Omron CX-Programmer project NewProject (CX-Programmer 9.51)

# PLC NewPLC1: CP1H XA

## Global symbols (name address type ; comment)
10.00 BOOL  ; internal input/hold bit
0.00 BOOL  ; input
100.00 BOOL  ; output

## Program NewProgram1 (cyclic task 0)

### Section Section1

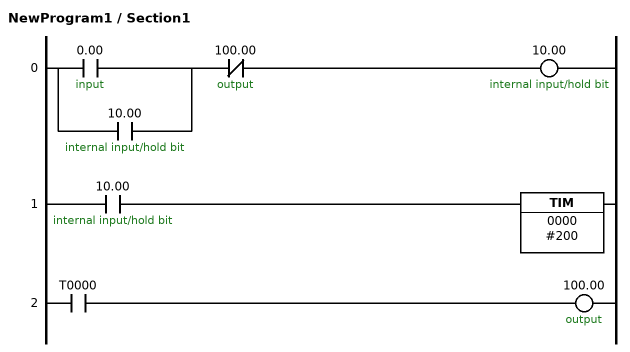
; rung 0
LD 0.00  ; input
OR 10.00  ; internal input/hold bit
ANDNOT 100.00  ; output
OUT 10.00  ; internal input/hold bit
; rung 1
LD 10.00  ; internal input/hold bit
TIM 0000 #200
; rung 2
LD T0000
OUT 100.00  ; output

### Section END
; rung 0
END(001)